    Win32ErrorCodes.ERROR_DS_GLOBAL_CANT_HAVE_LOCAL_MEMBER:
        Win32ErrorCodeDescription := 'A global group cannot have a local group as a member.';
    Win32ErrorCodes.ERROR_DS_GLOBAL_CANT_HAVE_UNIVERSAL_MEMBER:
        Win32ErrorCodeDescription := 'A global group cannot have a universal group as a member.';
    Win32ErrorCodes.ERROR_DS_UNIVERSAL_CANT_HAVE_LOCAL_MEMBER:
        Win32ErrorCodeDescription := 'A universal group cannot have a local group as a member.';
    Win32ErrorCodes.ERROR_DS_GLOBAL_CANT_HAVE_CROSSDOMAIN_MEMBER:
        Win32ErrorCodeDescription := 'A global group cannot have a cross-domain member.';
    Win32ErrorCodes.ERROR_DS_LOCAL_CANT_HAVE_CROSSDOMAIN_LOCAL_MEMBER:
        Win32ErrorCodeDescription :=
            'A local group cannot have another cross-domain local group as a member.';
    Win32ErrorCodes.ERROR_DS_HAVE_PRIMARY_MEMBERS:
        Win32ErrorCodeDescription :=
            'A group with primary members cannot change to a security-disabled group.';
    Win32ErrorCodes.ERROR_DS_STRING_SD_CONVERSION_FAILED:
        Win32ErrorCodeDescription :=
            'The schema cache load failed to convert the string default SD on a class-schema object.';
    Win32ErrorCodes.ERROR_DS_NAMING_MASTER_GC:
        Win32ErrorCodeDescription := 'Only DSAs configured to be Global Catalog servers should be allowed to hold the Domain Naming Master FSMO role. (Applies only to Windows 2000 servers)';
    Win32ErrorCodes.ERROR_DS_LOOKUP_FAILURE:
        Win32ErrorCodeDescription :=
            'The DSA operation is unable to proceed because of a DNS lookup failure.';
    Win32ErrorCodes.ERROR_DS_COULDNT_UPDATE_SPNS:
        Win32ErrorCodeDescription := 'While processing a change to the DNS Host Name for an object, the Service Principal Name values could not be kept in sync.';
    Win32ErrorCodes.ERROR_DS_CANT_RETRIEVE_SD:
        Win32ErrorCodeDescription := 'The Security Descriptor attribute could not be read.';
    Win32ErrorCodes.ERROR_DS_KEY_NOT_UNIQUE:
        Win32ErrorCodeDescription :=
            'The object requested was not found, but an object with that key was found.';
    Win32ErrorCodes.ERROR_DS_WRONG_LINKED_ATT_SYNTAX:
        Win32ErrorCodeDescription := 'The syntax of the linked attributed being added is incorrect. Forward links can only have syntax 2.5.5.1, 2.5.5.7, and 2.5.5.14, and backlinks can only have syntax 2.5.5.1.';
    Win32ErrorCodes.ERROR_DS_SAM_NEED_BOOTKEY_PASSWORD:
        Win32ErrorCodeDescription := 'Security Account Manager needs to get the boot password.';
    Win32ErrorCodes.ERROR_DS_SAM_NEED_BOOTKEY_FLOPPY:
        Win32ErrorCodeDescription :=
            'Security Account Manager needs to get the boot key from floppy disk.';
    Win32ErrorCodes.ERROR_DS_CANT_START:
        Win32ErrorCodeDescription := 'Directory Service cannot start.';
    Win32ErrorCodes.ERROR_DS_INIT_FAILURE:
        Win32ErrorCodeDescription := 'Directory Services could not start.';
    Win32ErrorCodes.ERROR_DS_NO_PKT_PRIVACY_ON_CONNECTION:
        Win32ErrorCodeDescription :=
            'The connection between client and server requires packet privacy or better.';
    Win32ErrorCodes.ERROR_DS_SOURCE_DOMAIN_IN_FOREST:
        Win32ErrorCodeDescription :=
            'The source domain may not be in the same forest as destination.';
    Win32ErrorCodes.ERROR_DS_DESTINATION_DOMAIN_NOT_IN_FOREST:
        Win32ErrorCodeDescription := 'The destination domain must be in the forest.';
    Win32ErrorCodes.ERROR_DS_DESTINATION_AUDITING_NOT_ENABLED:
        Win32ErrorCodeDescription :=
            'The operation requires that destination domain auditing be enabled.';
    Win32ErrorCodes.ERROR_DS_CANT_FIND_DC_FOR_SRC_DOMAIN:
        Win32ErrorCodeDescription := 'The operation couldnt locate a DC for the source domain.';
    Win32ErrorCodes.ERROR_DS_SRC_OBJ_NOT_GROUP_OR_USER:
        Win32ErrorCodeDescription := 'The source object must be a group or user.';
    Win32ErrorCodes.ERROR_DS_SRC_SID_EXISTS_IN_FOREST:
        Win32ErrorCodeDescription :=
            'The source objects SID already exists in destination forest.';
    Win32ErrorCodes.ERROR_DS_SRC_AND_DST_OBJECT_CLASS_MISMATCH:
        Win32ErrorCodeDescription := 'The source and destination object must be of the same type.';
    Win32ErrorCodes.ERROR_SAM_INIT_FAILURE:
        Win32ErrorCodeDescription := 'Security Accounts Manager initialization failed because of the following error: %1. Error Status: 0x%2. Click OK to shut down the system and reboot into Safe Mode. Check the event log for detailed information.';
    Win32ErrorCodes.ERROR_DS_DRA_SCHEMA_INFO_SHIP:
        Win32ErrorCodeDescription :=
            'Schema information could not be included in the replication request.';
    Win32ErrorCodes.ERROR_DS_DRA_SCHEMA_CONFLICT:
        Win32ErrorCodeDescription :=
            'The replication operation could not be completed due to a schema incompatibility.';
    Win32ErrorCodes.ERROR_DS_DRA_EARLIER_SCHEMA_CONLICT:
        Win32ErrorCodeDescription := 'The replication operation could not be completed due to a previous schema incompatibility.';
    Win32ErrorCodes.ERROR_DS_DRA_OBJ_NC_MISMATCH:
        Win32ErrorCodeDescription := 'The replication update could not be applied because either the source or the destination has not yet received information regarding a recent cross-domain move operation.';
    Win32ErrorCodes.ERROR_DS_NC_STILL_HAS_DSAS:
        Win32ErrorCodeDescription := 'The requested domain could not be deleted because there exist domain controllers that still host this domain.';
    Win32ErrorCodes.ERROR_DS_GC_REQUIRED:
        Win32ErrorCodeDescription :=
            'The requested operation can be performed only on a global catalog server.';
    Win32ErrorCodes.ERROR_DS_LOCAL_MEMBER_OF_LOCAL_ONLY:
        Win32ErrorCodeDescription :=
            'A local group can only be a member of other local groups in the same domain.';
    Win32ErrorCodes.ERROR_DS_NO_FPO_IN_UNIVERSAL_GROUPS:
        Win32ErrorCodeDescription :=
            'Foreign security principals cannot be members of universal groups.';
    Win32ErrorCodes.ERROR_DS_CANT_ADD_TO_GC:
        Win32ErrorCodeDescription :=
            'The attribute is not allowed to be replicated to the GC because of security reasons.';
    Win32ErrorCodes.ERROR_DS_NO_CHECKPOINT_WITH_PDC:
        Win32ErrorCodeDescription := 'The checkpoint with the PDC could not be taken because there are too many modifications being processed currently.';
    Win32ErrorCodes.ERROR_DS_SOURCE_AUDITING_NOT_ENABLED:
        Win32ErrorCodeDescription :=
            'The operation requires that source domain auditing be enabled.';
    Win32ErrorCodes.ERROR_DS_CANT_CREATE_IN_NONDOMAIN_NC:
        Win32ErrorCodeDescription :=
            'Security principal objects can only be created inside domain naming contexts.';
    Win32ErrorCodes.ERROR_DS_INVALID_NAME_FOR_SPN:
        Win32ErrorCodeDescription := 'A Service Principal Name (SPN) could not be constructed because the provided hostname is not in the necessary format.';
    Win32ErrorCodes.ERROR_DS_FILTER_USES_CONTRUCTED_ATTRS:
        Win32ErrorCodeDescription := 'A Filter was passed that uses constructed attributes.';
    Win32ErrorCodes.ERROR_DS_UNICODEPWD_NOT_IN_QUOTES:
        Win32ErrorCodeDescription :=
            'The unicodePwd attribute value must be enclosed in double quotes.';
    Win32ErrorCodes.ERROR_DS_MACHINE_ACCOUNT_QUOTA_EXCEEDED:
        Win32ErrorCodeDescription := 'Your computer could not be joined to the domain. You have exceeded the maximum number of computer accounts you are allowed to create in this domain. Contact your system administrator to have this limit reset or increased.';
    Win32ErrorCodes.ERROR_DS_MUST_BE_RUN_ON_DST_DC:
        Win32ErrorCodeDescription :=
            'For security reasons, the operation must be run on the destination DC.';
    Win32ErrorCodes.ERROR_DS_SRC_DC_MUST_BE_SP4_OR_GREATER:
        Win32ErrorCodeDescription :=
            'For security reasons, the source DC must be NT4SP4 or greater.';
    Win32ErrorCodes.ERROR_DS_CANT_TREE_DELETE_CRITICAL_OBJ:
        Win32ErrorCodeDescription := 'Critical Directory Service System objects cannot be deleted during tree delete operations. The tree delete may have been partially performed.';
    Win32ErrorCodes.ERROR_DS_INIT_FAILURE_CONSOLE:
        Win32ErrorCodeDescription := 'Directory Services could not start because of the following error: %1. Error Status: 0x%2. Please click OK to shutdown the system. You can use the recovery console to diagnose the system further.';
    Win32ErrorCodes.ERROR_DS_SAM_INIT_FAILURE_CONSOLE:
        Win32ErrorCodeDescription := 'Security Accounts Manager initialization failed because of the following error: %1. Error Status: 0x%2. Please click OK to shutdown the system. You can use the recovery console to diagnose the system further.';
    Win32ErrorCodes.ERROR_DS_FOREST_VERSION_TOO_HIGH:
        Win32ErrorCodeDescription := 'This version of Windows is too old to support the current directory forest behavior. You must upgrade the operating system on this server before it can become a domain controller in this forest.';
    Win32ErrorCodes.ERROR_DS_DOMAIN_VERSION_TOO_HIGH:
        Win32ErrorCodeDescription := 'This version of Windows is too old to support the current domain behavior. You must upgrade the operating system on this server before it can become a domain controller in this domain.';
    Win32ErrorCodes.ERROR_DS_FOREST_VERSION_TOO_LOW:
        Win32ErrorCodeDescription := 'This version of Windows no longer supports the behavior version in use in this directory forest. You must advance the forest behavior version before this server can become a domain controller in the forest.';
    Win32ErrorCodes.ERROR_DS_DOMAIN_VERSION_TOO_LOW:
        Win32ErrorCodeDescription := 'This version of Windows no longer supports the behavior version in use in this domain. You must advance the domain behavior version before this server can become a domain controller in the domain.';
    Win32ErrorCodes.ERROR_DS_INCOMPATIBLE_VERSION:
        Win32ErrorCodeDescription :=
            'The version of Windows is incompatible with the behavior version of the domain or forest.';
    Win32ErrorCodes.ERROR_DS_LOW_DSA_VERSION:
        Win32ErrorCodeDescription := 'The behavior version cannot be increased to the requested value because Domain Controllers still exist with versions lower than the requested value.';
    Win32ErrorCodes.ERROR_DS_NO_BEHAVIOR_VERSION_IN_MIXEDDOMAIN:
        Win32ErrorCodeDescription := 'The behavior version value cannot be increased while the domain is still in mixed domain mode. You must first change the domain to native mode before increasing the behavior version.';
    Win32ErrorCodes.ERROR_DS_NOT_SUPPORTED_SORT_ORDER:
        Win32ErrorCodeDescription := 'The sort order requested is not supported.';
    Win32ErrorCodes.ERROR_DS_NAME_NOT_UNIQUE:
        Win32ErrorCodeDescription := 'Found an object with a non unique name.';
    Win32ErrorCodes.ERROR_DS_MACHINE_ACCOUNT_CREATED_PRENT4:
        Win32ErrorCodeDescription :=
            'The machine account was created pre-NT4. The account needs to be recreated.';
    Win32ErrorCodes.ERROR_DS_OUT_OF_VERSION_STORE:
        Win32ErrorCodeDescription := 'The database is out of version store.';
    Win32ErrorCodes.ERROR_DS_INCOMPATIBLE_CONTROLS_USED:
        Win32ErrorCodeDescription :=
            'Unable to continue operation because multiple conflicting controls were used.';
    Win32ErrorCodes.ERROR_DS_NO_REF_DOMAIN:
        Win32ErrorCodeDescription :=
            'Unable to find a valid security descriptor reference domain for this partition.';
    Win32ErrorCodes.ERROR_DS_RESERVED_LINK_ID:
        Win32ErrorCodeDescription := 'Schema update failed: The link identifier is reserved.';
    Win32ErrorCodes.ERROR_DS_LINK_ID_NOT_AVAILABLE:
        Win32ErrorCodeDescription :=
            'Schema update failed: There are no link identifiers available.';
    Win32ErrorCodes.ERROR_DS_AG_CANT_HAVE_UNIVERSAL_MEMBER:
        Win32ErrorCodeDescription :=
            'An account group can not have a universal group as a member.';
    Win32ErrorCodes.ERROR_DS_MODIFYDN_DISALLOWED_BY_INSTANCE_TYPE:
        Win32ErrorCodeDescription :=
            'Rename or move operations on naming context heads or read-only objects are not allowed.';
    Win32ErrorCodes.ERROR_DS_NO_OBJECT_MOVE_IN_SCHEMA_NC:
        Win32ErrorCodeDescription :=
            'Move operations on objects in the schema naming context are not allowed.';
    Win32ErrorCodes.ERROR_DS_MODIFYDN_DISALLOWED_BY_FLAG:
        Win32ErrorCodeDescription := 'A system flag has been set on the object and does not allow the object to be moved or renamed.';
    Win32ErrorCodes.ERROR_DS_MODIFYDN_WRONG_GRANDPARENT:
        Win32ErrorCodeDescription := 'This object is not allowed to change its grandparent container. Moves are not forbidden on this object, but are restricted to sibling containers.';
    Win32ErrorCodes.ERROR_DS_NAME_ERROR_TRUST_REFERRAL:
        Win32ErrorCodeDescription :=
            'Unable to resolve completely, a referral to another forest is generated.';
    Win32ErrorCodes.ERROR_NOT_SUPPORTED_ON_STANDARD_SERVER:
        Win32ErrorCodeDescription := 'The requested action is not supported on standard server.';
    Win32ErrorCodes.ERROR_DS_CANT_ACCESS_REMOTE_PART_OF_AD:
        Win32ErrorCodeDescription := 'Could not access a partition of the Active Directory located on a remote server. Make sure at least one server is running for the partition in question.';
    Win32ErrorCodes.ERROR_DS_CR_IMPOSSIBLE_TO_VALIDATE_V2:
        Win32ErrorCodeDescription := 'The directory cant validate the proposed naming context (or partition) name because it doesnt hold a replica nor can it contact a replica of the naming context above the proposed naming context.';
    Win32ErrorCodes.ERROR_DS_THREAD_LIMIT_EXCEEDED:
        Win32ErrorCodeDescription := 'The thread limit for this request was exceeded.';
    Win32ErrorCodes.ERROR_DS_NOT_CLOSEST:
        Win32ErrorCodeDescription := 'The Global catalog server is not in the closet site.';
    Win32ErrorCodes.DNS_ERROR_RCODE_FORMAT_ERROR:
        Win32ErrorCodeDescription := 'DNS server unable to interpret format.';
    Win32ErrorCodes.DNS_ERROR_RCODE_SERVER_FAILURE:
        Win32ErrorCodeDescription := 'DNS server failure.';
    Win32ErrorCodes.DNS_ERROR_RCODE_NAME_ERROR:
        Win32ErrorCodeDescription := 'DNS name does not exist.';
    Win32ErrorCodes.DNS_ERROR_RCODE_NOT_IMPLEMENTED:
        Win32ErrorCodeDescription := 'DNS request not supported by name server.';
    Win32ErrorCodes.DNS_ERROR_RCODE_REFUSED:
        Win32ErrorCodeDescription := 'DNS operation refused.';
    Win32ErrorCodes.DNS_ERROR_RCODE_YXDOMAIN:
        Win32ErrorCodeDescription := 'DNS name that ought not exist, does exist.';
    Win32ErrorCodes.DNS_ERROR_RCODE_YXRRSET:
        Win32ErrorCodeDescription := 'DNS RR set that ought not exist, does exist.';
    Win32ErrorCodes.DNS_ERROR_RCODE_NXRRSET:
        Win32ErrorCodeDescription := 'DNS RR set that ought to exist, does not exist.';
    Win32ErrorCodes.DNS_ERROR_RCODE_NOTAUTH:
        Win32ErrorCodeDescription := 'DNS server not authoritative for zone.';
    Win32ErrorCodes.DNS_ERROR_RCODE_NOTZONE:
        Win32ErrorCodeDescription := 'DNS name in update or prereq is not in zone.';
    Win32ErrorCodes.DNS_ERROR_RCODE_BADSIG:
        Win32ErrorCodeDescription := 'DNS signature failed to verify.';
    Win32ErrorCodes.DNS_ERROR_RCODE_BADKEY:
        Win32ErrorCodeDescription := 'DNS bad key.';
    Win32ErrorCodes.DNS_ERROR_RCODE_BADTIME:
        Win32ErrorCodeDescription := 'DNS signature validity expired.';
    Win32ErrorCodes.DNS_INFO_NO_RECORDS:
        Win32ErrorCodeDescription := 'No records found for given DNS query.';
    Win32ErrorCodes.DNS_ERROR_BAD_PACKET:
        Win32ErrorCodeDescription := 'Bad DNS packet.';
    Win32ErrorCodes.DNS_ERROR_NO_PACKET:
        Win32ErrorCodeDescription := 'No DNS packet.';
    Win32ErrorCodes.DNS_ERROR_RCODE:
        Win32ErrorCodeDescription := 'DNS error, check rcode.';
    Win32ErrorCodes.DNS_ERROR_UNSECURE_PACKET:
        Win32ErrorCodeDescription := 'Unsecured DNS packet.';
    Win32ErrorCodes.DNS_ERROR_INVALID_TYPE:
        Win32ErrorCodeDescription := 'Invalid DNS type.';
    Win32ErrorCodes.DNS_ERROR_INVALID_IP_ADDRESS:
        Win32ErrorCodeDescription := 'Invalid IP address.';
    Win32ErrorCodes.DNS_ERROR_INVALID_PROPERTY:
        Win32ErrorCodeDescription := 'Invalid property.';
    Win32ErrorCodes.DNS_ERROR_TRY_AGAIN_LATER:
        Win32ErrorCodeDescription := 'Try DNS operation again later.';
    Win32ErrorCodes.DNS_ERROR_NOT_UNIQUE:
        Win32ErrorCodeDescription := 'Record for given name and type is not unique.';
    Win32ErrorCodes.DNS_ERROR_NON_RFC_NAME:
        Win32ErrorCodeDescription := 'DNS name does not comply with RFC specifications.';
    Win32ErrorCodes.DNS_STATUS_FQDN:
        Win32ErrorCodeDescription := 'DNS name is a fully-qualified DNS name.';
    Win32ErrorCodes.DNS_STATUS_DOTTED_NAME:
        Win32ErrorCodeDescription := 'DNS name is dotted (multi-label).';
    Win32ErrorCodes.DNS_STATUS_SINGLE_PART_NAME:
        Win32ErrorCodeDescription := 'DNS name is a single-part name.';
    Win32ErrorCodes.DNS_ERROR_INVALID_NAME_CHAR:
        Win32ErrorCodeDescription := 'DSN name contains an invalid character.';
    Win32ErrorCodes.DNS_ERROR_NUMERIC_NAME:
        Win32ErrorCodeDescription := 'DNS name is entirely numeric.';
    Win32ErrorCodes.DNS_ERROR_ZONE_DOES_NOT_EXIST:
        Win32ErrorCodeDescription := 'DNS zone does not exist.';
    Win32ErrorCodes.DNS_ERROR_NO_ZONE_INFO:
        Win32ErrorCodeDescription := 'DNS zone information not available.';
    Win32ErrorCodes.DNS_ERROR_INVALID_ZONE_OPERATION:
        Win32ErrorCodeDescription := 'Invalid operation for DNS zone.';
    Win32ErrorCodes.DNS_ERROR_ZONE_CONFIGURATION_ERROR:
        Win32ErrorCodeDescription := 'Invalid DNS zone configuration.';
    Win32ErrorCodes.DNS_ERROR_ZONE_HAS_NO_SOA_RECORD:
        Win32ErrorCodeDescription := 'DNS zone has no start of authority (SOA) record.';
    Win32ErrorCodes.DNS_ERROR_ZONE_HAS_NO_NS_RECORDS:
        Win32ErrorCodeDescription := 'DNS zone has no name server (NS) record.';
    Win32ErrorCodes.DNS_ERROR_ZONE_LOCKED:
        Win32ErrorCodeDescription := 'DNS zone is locked.';
    Win32ErrorCodes.DNS_ERROR_ZONE_CREATION_FAILED:
        Win32ErrorCodeDescription := 'DNS zone creation failed.';
    Win32ErrorCodes.DNS_ERROR_ZONE_ALREADY_EXISTS:
        Win32ErrorCodeDescription := 'DNS zone already exists.';
    Win32ErrorCodes.DNS_ERROR_AUTOZONE_ALREADY_EXISTS:
        Win32ErrorCodeDescription := 'DNS automatic zone already exists.';
    Win32ErrorCodes.DNS_ERROR_INVALID_ZONE_TYPE:
        Win32ErrorCodeDescription := 'Invalid DNS zone type.';
    Win32ErrorCodes.DNS_ERROR_SECONDARY_REQUIRES_MASTER_IP:
        Win32ErrorCodeDescription := 'Secondary DNS zone requires master IP address.';
    Win32ErrorCodes.DNS_ERROR_ZONE_NOT_SECONDARY:
        Win32ErrorCodeDescription := 'DNS zone not secondary.';
    Win32ErrorCodes.DNS_ERROR_NEED_SECONDARY_ADDRESSES:
        Win32ErrorCodeDescription := 'Need secondary IP address.';
    Win32ErrorCodes.DNS_ERROR_WINS_INIT_FAILED:
        Win32ErrorCodeDescription := 'WINS initialization failed.';
    Win32ErrorCodes.DNS_ERROR_NEED_WINS_SERVERS:
        Win32ErrorCodeDescription := 'Need WINS servers.';
    Win32ErrorCodes.DNS_ERROR_NBSTAT_INIT_FAILED:
        Win32ErrorCodeDescription := 'NBTSTAT initialization call failed.';
    Win32ErrorCodes.DNS_ERROR_SOA_DELETE_INVALID:
        Win32ErrorCodeDescription := 'Invalid delete of start of authority (SOA)';
    Win32ErrorCodes.DNS_ERROR_FORWARDER_ALREADY_EXISTS:
        Win32ErrorCodeDescription := 'A conditional forwarding zone already exists for that name.';
    Win32ErrorCodes.DNS_ERROR_PRIMARY_REQUIRES_DATAFILE:
        Win32ErrorCodeDescription := 'Primary DNS zone requires datafile.';
    Win32ErrorCodes.DNS_ERROR_INVALID_DATAFILE_NAME:
        Win32ErrorCodeDescription := 'Invalid datafile name for DNS zone.';
    Win32ErrorCodes.DNS_ERROR_DATAFILE_OPEN_FAILURE:
        Win32ErrorCodeDescription := 'Failed to open datafile for DNS zone.';
    Win32ErrorCodes.DNS_ERROR_FILE_WRITEBACK_FAILED:
        Win32ErrorCodeDescription := 'Failed to write datafile for DNS zone.';
    Win32ErrorCodes.DNS_ERROR_DATAFILE_PARSING:
        Win32ErrorCodeDescription := 'Failure while reading datafile for DNS zone.';
    Win32ErrorCodes.DNS_ERROR_RECORD_DOES_NOT_EXIST:
        Win32ErrorCodeDescription := 'DNS record does not exist.';
    Win32ErrorCodes.DNS_ERROR_RECORD_FORMAT:
        Win32ErrorCodeDescription := 'DNS record format error.';
    Win32ErrorCodes.DNS_ERROR_NODE_CREATION_FAILED:
        Win32ErrorCodeDescription := 'Node creation failure in DNS.';
    Win32ErrorCodes.DNS_ERROR_UNKNOWN_RECORD_TYPE:
        Win32ErrorCodeDescription := 'Unknown DNS record type.';
    Win32ErrorCodes.DNS_ERROR_RECORD_TIMED_OUT:
        Win32ErrorCodeDescription := 'DNS record timed out.';
    Win32ErrorCodes.DNS_ERROR_NAME_NOT_IN_ZONE:
        Win32ErrorCodeDescription := 'Name not in DNS zone.';
    Win32ErrorCodes.DNS_ERROR_CNAME_LOOP:
        Win32ErrorCodeDescription := 'CNAME loop detected.';
    Win32ErrorCodes.DNS_ERROR_NODE_IS_CNAME:
        Win32ErrorCodeDescription := 'Node is a CNAME DNS record.';
    Win32ErrorCodes.DNS_ERROR_CNAME_COLLISION:
        Win32ErrorCodeDescription := 'A CNAME record already exists for given name.';
    Win32ErrorCodes.DNS_ERROR_RECORD_ONLY_AT_ZONE_ROOT:
        Win32ErrorCodeDescription := 'Record only at DNS zone root.';
    Win32ErrorCodes.DNS_ERROR_RECORD_ALREADY_EXISTS:
        Win32ErrorCodeDescription := 'DNS record already exists.';
    Win32ErrorCodes.DNS_ERROR_SECONDARY_DATA:
        Win32ErrorCodeDescription := 'Secondary DNS zone data error.';
    Win32ErrorCodes.DNS_ERROR_NO_CREATE_CACHE_DATA:
        Win32ErrorCodeDescription := 'Could not create DNS cache data.';
    Win32ErrorCodes.DNS_ERROR_NAME_DOES_NOT_EXIST:
        Win32ErrorCodeDescription := 'DNS name does not exist.';
    Win32ErrorCodes.DNS_WARNING_PTR_CREATE_FAILED:
        Win32ErrorCodeDescription := 'Could not create pointer (PTR) record.';
    Win32ErrorCodes.DNS_WARNING_DOMAIN_UNDELETED:
        Win32ErrorCodeDescription := 'DNS domain was undeleted.';
    Win32ErrorCodes.DNS_ERROR_DS_UNAVAILABLE:
        Win32ErrorCodeDescription := 'The directory service is unavailable.';
    Win32ErrorCodes.DNS_ERROR_DS_ZONE_ALREADY_EXISTS:
        Win32ErrorCodeDescription := 'DNS zone already exists in the directory service.';
    Win32ErrorCodes.DNS_ERROR_NO_BOOTFILE_IF_DS_ZONE:
        Win32ErrorCodeDescription := 'DNS server not creating or reading the boot file for the directory service integrated DNS zone.';
    Win32ErrorCodes.DNS_INFO_AXFR_COMPLETE:
        Win32ErrorCodeDescription := 'DNS AXFR (zone transfer) complete.';
    Win32ErrorCodes.DNS_ERROR_AXFR:
        Win32ErrorCodeDescription := 'DNS zone transfer failed.';
    Win32ErrorCodes.DNS_INFO_ADDED_LOCAL_WINS:
        Win32ErrorCodeDescription := 'Added local WINS server.';
    Win32ErrorCodes.DNS_STATUS_CONTINUE_NEEDED:
        Win32ErrorCodeDescription := 'Secure update call needs to continue update request.';
    Win32ErrorCodes.DNS_ERROR_NO_TCPIP:
        Win32ErrorCodeDescription := 'TCP/IP network protocol not installed.';
    Win32ErrorCodes.DNS_ERROR_NO_DNS_SERVERS:
        Win32ErrorCodeDescription := 'No DNS servers configured for local system.';
    Win32ErrorCodes.DNS_ERROR_DP_DOES_NOT_EXIST:
        Win32ErrorCodeDescription := 'The specified directory partition does not exist.';
    Win32ErrorCodes.DNS_ERROR_DP_ALREADY_EXISTS:
        Win32ErrorCodeDescription := 'The specified directory partition already exists.';
    Win32ErrorCodes.DNS_ERROR_DP_NOT_ENLISTED:
        Win32ErrorCodeDescription :=
            'The DS is not enlisted in the specified directory partition.';
    Win32ErrorCodes.DNS_ERROR_DP_ALREADY_ENLISTED:
        Win32ErrorCodeDescription :=
            'The DS is already enlisted in the specified directory partition.';
    Win32ErrorCodes.WSAEINTR:
        Win32ErrorCodeDescription :=
            'A blocking operation was interrupted by a call to WSACancelBlockingCall.';
    Win32ErrorCodes.WSAEBADF:
        Win32ErrorCodeDescription := 'The file handle supplied is not valid.';
    Win32ErrorCodes.WSAEACCES:
        Win32ErrorCodeDescription :=
            'An attempt was made to access a socket in a way forbidden by its access permissions.';
    Win32ErrorCodes.WSAEFAULT:
        Win32ErrorCodeDescription := 'The system detected an invalid pointer address in attempting to use a pointer argument in a call.';
    Win32ErrorCodes.WSAEINVAL:
        Win32ErrorCodeDescription := 'An invalid argument was supplied.';
    Win32ErrorCodes.WSAEMFILE:
        Win32ErrorCodeDescription := 'Too many open sockets.';
    Win32ErrorCodes.WSAEWOULDBLOCK:
        Win32ErrorCodeDescription :=
            'A non-blocking socket operation could not be completed immediately.';
    Win32ErrorCodes.WSAEINPROGRESS:
        Win32ErrorCodeDescription := 'A blocking operation is currently executing.';
    Win32ErrorCodes.WSAEALREADY:
        Win32ErrorCodeDescription := 'An operation was attempted on a non-blocking socket that already had an operation in progress.';
    Win32ErrorCodes.WSAENOTSOCK:
        Win32ErrorCodeDescription :=
            'An operation was attempted on something that is not a socket.';
    Win32ErrorCodes.WSAEDESTADDRREQ:
        Win32ErrorCodeDescription :=
            'A required address was omitted from an operation on a socket.';
    Win32ErrorCodes.WSAEMSGSIZE:
        Win32ErrorCodeDescription := 'A message sent on a datagram socket was larger than the internal message buffer or some other network limit, or the buffer used to receive a datagram into was smaller than the datagram itself.';
    Win32ErrorCodes.WSAEPROTOTYPE:
        Win32ErrorCodeDescription := 'A protocol was specified in the socket function call that does not support the semantics of the socket type requested.';
    Win32ErrorCodes.WSAENOPROTOOPT:
        Win32ErrorCodeDescription := 'An unknown, invalid, or unsupported option or level was specified in a getsockopt or setsockopt call.';
    Win32ErrorCodes.WSAEPROTONOSUPPORT:
        Win32ErrorCodeDescription := 'The requested protocol has not been configured into the system, or no implementation for it exists.';
    Win32ErrorCodes.WSAESOCKTNOSUPPORT:
        Win32ErrorCodeDescription :=
            'The support for the specified socket type does not exist in this address family.';
    Win32ErrorCodes.WSAEOPNOTSUPP:
        Win32ErrorCodeDescription :=
            'The attempted operation is not supported for the type of object referenced.';
    Win32ErrorCodes.WSAEPFNOSUPPORT:
        Win32ErrorCodeDescription := 'The protocol family has not been configured into the system or no implementation for it exists.';
    Win32ErrorCodes.WSAEAFNOSUPPORT:
        Win32ErrorCodeDescription :=
            'An address incompatible with the requested protocol was used.';
    Win32ErrorCodes.WSAEADDRINUSE:
        Win32ErrorCodeDescription := 'Only one usage of each socket address (protocol/network address/port) is normally permitted.';
    Win32ErrorCodes.WSAEADDRNOTAVAIL:
        Win32ErrorCodeDescription := 'The requested address is not valid in its context.';
    Win32ErrorCodes.WSAENETDOWN:
        Win32ErrorCodeDescription := 'A socket operation encountered a dead network.';
    Win32ErrorCodes.WSAENETUNREACH:
        Win32ErrorCodeDescription := 'A socket operation was attempted to an unreachable network.';
    Win32ErrorCodes.WSAENETRESET:
        Win32ErrorCodeDescription := 'The connection has been broken due to keep-alive activity detecting a failure while the operation was in progress.';
    Win32ErrorCodes.WSAECONNABORTED:
        Win32ErrorCodeDescription :=
            'An established connection was aborted by the software in your host machine.';
    Win32ErrorCodes.WSAECONNRESET:
        Win32ErrorCodeDescription :=
            'An existing connection was forcibly closed by the remote host.';
    Win32ErrorCodes.WSAENOBUFS:
        Win32ErrorCodeDescription := 'An operation on a socket could not be performed because the system lacked sufficient buffer space or because a queue was full.';
    Win32ErrorCodes.WSAEISCONN:
        Win32ErrorCodeDescription := 'A connect request was made on an already connected socket.';
    Win32ErrorCodes.WSAENOTCONN:
        Win32ErrorCodeDescription := 'A request to send or receive data was disallowed because the socket is not connected and (when sending on a datagram socket using a sendto call) no address was supplied.';
    Win32ErrorCodes.WSAESHUTDOWN:
        Win32ErrorCodeDescription := 'A request to send or receive data was disallowed because the socket had already been shut down in that direction with a previous shutdown call.';
    Win32ErrorCodes.WSAETOOMANYREFS:
        Win32ErrorCodeDescription := 'Too many references to some kernel object.';
    Win32ErrorCodes.WSAETIMEDOUT:
        Win32ErrorCodeDescription := 'A connection attempt failed because the connected party did not properly respond after a period of time, or established connection failed because connected host has failed to respond.';
    Win32ErrorCodes.WSAECONNREFUSED:
        Win32ErrorCodeDescription :=
            'No connection could be made because the target machine actively refused it.';
    Win32ErrorCodes.WSAELOOP:
        Win32ErrorCodeDescription := 'Cannot translate name.';
    Win32ErrorCodes.WSAENAMETOOLONG:
        Win32ErrorCodeDescription := 'Name component or name was too long.';
    Win32ErrorCodes.WSAEHOSTDOWN:
        Win32ErrorCodeDescription :=
            'A socket operation failed because the destination host was down.';
    Win32ErrorCodes.WSAEHOSTUNREACH:
        Win32ErrorCodeDescription := 'A socket operation was attempted to an unreachable host.';
    Win32ErrorCodes.WSAENOTEMPTY:
        Win32ErrorCodeDescription := 'Cannot remove a directory that is not empty.';
    Win32ErrorCodes.WSAEPROCLIM:
        Win32ErrorCodeDescription := 'A Windows Sockets implementation may have a limit on the number of applications that may use it simultaneously.';
    Win32ErrorCodes.WSAEUSERS:
        Win32ErrorCodeDescription := 'Ran out of quota.';
    Win32ErrorCodes.WSAEDQUOT:
        Win32ErrorCodeDescription := 'Ran out of disk quota.';
    Win32ErrorCodes.WSAESTALE:
        Win32ErrorCodeDescription := 'File handle reference is no longer available.';
    Win32ErrorCodes.WSAEREMOTE:
        Win32ErrorCodeDescription := 'Item is not available locally.';
    Win32ErrorCodes.WSASYSNOTREADY:
        Win32ErrorCodeDescription := 'WSAStartup cannot function at this time because the underlying system it uses to provide network services is currently unavailable.';
    Win32ErrorCodes.WSAVERNOTSUPPORTED:
        Win32ErrorCodeDescription := 'The Windows Sockets version requested is not supported.';
    Win32ErrorCodes.WSANOTINITIALISED:
        Win32ErrorCodeDescription :=
            'Either the application has not called WSAStartup, or WSAStartup failed.';
    Win32ErrorCodes.WSAEDISCON:
        Win32ErrorCodeDescription := 'Returned by WSARecv or WSARecvFrom to indicate the remote party has initiated a graceful shutdown sequence.';
    Win32ErrorCodes.WSAENOMORE:
        Win32ErrorCodeDescription := 'No more results can be returned by WSALookupServiceNext.';
    Win32ErrorCodes.WSAECANCELLED:
        Win32ErrorCodeDescription := 'A call to WSALookupServiceEnd was made while this call was still processing. The call has been canceled.';
    Win32ErrorCodes.WSAEINVALIDPROCTABLE:
        Win32ErrorCodeDescription := 'The procedure call table is invalid.';
    Win32ErrorCodes.WSAEINVALIDPROVIDER:
        Win32ErrorCodeDescription := 'The requested service provider is invalid.';
    Win32ErrorCodes.WSAEPROVIDERFAILEDINIT:
        Win32ErrorCodeDescription :=
            'The requested service provider could not be loaded or initialized.';
    Win32ErrorCodes.WSASYSCALLFAILURE:
        Win32ErrorCodeDescription := 'A system call that should never fail has failed.';
    Win32ErrorCodes.WSASERVICE_NOT_FOUND:
        Win32ErrorCodeDescription :=
            'No such service is known. The service cannot be found in the specified name space.';
    Win32ErrorCodes.WSATYPE_NOT_FOUND:
        Win32ErrorCodeDescription := 'The specified class was not found.';
    Win32ErrorCodes.WSA_E_NO_MORE:
        Win32ErrorCodeDescription := 'No more results can be returned by WSALookupServiceNext.';
    Win32ErrorCodes.WSA_E_CANCELLED:
        Win32ErrorCodeDescription := 'A call to WSALookupServiceEnd was made while this call was still processing. The call has been canceled.';
    Win32ErrorCodes.WSAEREFUSED:
        Win32ErrorCodeDescription := 'A database query failed because it was actively refused.';
    Win32ErrorCodes.WSAHOST_NOT_FOUND:
        Win32ErrorCodeDescription := 'No such host is known.';
    Win32ErrorCodes.WSATRY_AGAIN:
        Win32ErrorCodeDescription := 'This is usually a temporary error during hostname resolution and means that the local server did not receive a response from an authoritative server.';
    Win32ErrorCodes.WSANO_RECOVERY:
        Win32ErrorCodeDescription := 'A non-recoverable error occurred during a database lookup.';
    Win32ErrorCodes.WSANO_DATA:
        Win32ErrorCodeDescription := 'The requested name is valid and was found in the database, but it does not have the correct associated data being resolved for.';
    Win32ErrorCodes.WSA_QOS_RECEIVERS:
        Win32ErrorCodeDescription := 'At least one reserve has arrived.';
    Win32ErrorCodes.WSA_QOS_SENDERS:
        Win32ErrorCodeDescription := 'At least one path has arrived.';
    Win32ErrorCodes.WSA_QOS_NO_SENDERS:
        Win32ErrorCodeDescription := 'There are no senders.';
    Win32ErrorCodes.WSA_QOS_NO_RECEIVERS:
        Win32ErrorCodeDescription := 'There are no receivers.';
    Win32ErrorCodes.WSA_QOS_REQUEST_CONFIRMED:
        Win32ErrorCodeDescription := 'Reserve has been confirmed.';
    Win32ErrorCodes.WSA_QOS_ADMISSION_FAILURE:
        Win32ErrorCodeDescription := 'Error due to lack of resources.';
    Win32ErrorCodes.WSA_QOS_POLICY_FAILURE:
        Win32ErrorCodeDescription := 'Rejected for administrative reasons - bad credentials.';
    Win32ErrorCodes.WSA_QOS_BAD_STYLE:
        Win32ErrorCodeDescription := 'Unknown or conflicting style.';
    Win32ErrorCodes.WSA_QOS_BAD_OBJECT:
        Win32ErrorCodeDescription :=
            'Problem with some part of the filterspec or providerspecific buffer in general.';
    Win32ErrorCodes.WSA_QOS_TRAFFIC_CTRL_ERROR:
        Win32ErrorCodeDescription := 'Problem with some part of the flowspec.';
    Win32ErrorCodes.WSA_QOS_GENERIC_ERROR:
        Win32ErrorCodeDescription := 'General QOS error.';
    Win32ErrorCodes.WSA_QOS_ESERVICETYPE:
        Win32ErrorCodeDescription :=
            'An invalid or unrecognized service type was found in the flowspec.';
    Win32ErrorCodes.WSA_QOS_EFLOWSPEC:
        Win32ErrorCodeDescription :=
            'An invalid or inconsistent flowspec was found in the QOS structure.';
    Win32ErrorCodes.WSA_QOS_EPROVSPECBUF:
        Win32ErrorCodeDescription := 'Invalid QOS provider-specific buffer.';
    Win32ErrorCodes.WSA_QOS_EFILTERSTYLE:
        Win32ErrorCodeDescription := 'An invalid QOS filter style was used.';
    Win32ErrorCodes.WSA_QOS_EFILTERTYPE:
        Win32ErrorCodeDescription := 'An invalid QOS filter type was used.';
    Win32ErrorCodes.WSA_QOS_EFILTERCOUNT:
        Win32ErrorCodeDescription :=
            'An incorrect number of QOS FILTERSPECs were specified in the FLOWDESCRIPTOR.';
    Win32ErrorCodes.WSA_QOS_EOBJLENGTH:
        Win32ErrorCodeDescription := 'An object with an invalid ObjectLength field was specified in the QOS provider-specific buffer.';
    Win32ErrorCodes.WSA_QOS_EFLOWCOUNT:
        Win32ErrorCodeDescription :=
            'An incorrect number of flow descriptors was specified in the QOS structure.';
    Win32ErrorCodes.WSA_QOS_EUNKNOWNPSOBJ:
        Win32ErrorCodeDescription :=
            'An unrecognized object was found in the QOS provider-specific buffer.';
    Win32ErrorCodes.WSA_QOS_EPOLICYOBJ:
        Win32ErrorCodeDescription :=
            'An invalid policy object was found in the QOS provider-specific buffer.';
    Win32ErrorCodes.WSA_QOS_EFLOWDESC:
        Win32ErrorCodeDescription :=
            'An invalid QOS flow descriptor was found in the flow descriptor list.';
    Win32ErrorCodes.WSA_QOS_EPSFLOWSPEC:
        Win32ErrorCodeDescription :=
            'An invalid or inconsistent flowspec was found in the QOS provider-specific buffer.';
    Win32ErrorCodes.WSA_QOS_EPSFILTERSPEC:
        Win32ErrorCodeDescription :=
            'An invalid FILTERSPEC was found in the QOS provider-specific buffer.';
    Win32ErrorCodes.WSA_QOS_ESDMODEOBJ:
        Win32ErrorCodeDescription :=
            'An invalid shape discard mode object was found in the QOS provider-specific buffer.';
    Win32ErrorCodes.WSA_QOS_ESHAPERATEOBJ:
        Win32ErrorCodeDescription :=
            'An invalid shaping rate object was found in the QOS provider-specific buffer.';
    Win32ErrorCodes.WSA_QOS_RESERVED_PETYPE:
        Win32ErrorCodeDescription :=
            'A reserved policy element was found in the QOS provider-specific buffer.';
    Win32ErrorCodes.ERROR_SXS_SECTION_NOT_FOUND:
        Win32ErrorCodeDescription :=
            'The requested section was not present in the activation context.';
    Win32ErrorCodes.ERROR_SXS_CANT_GEN_ACTCTX:
        Win32ErrorCodeDescription := 'This application has failed to start because the application configuration is incorrect. Reinstalling the application may fix this problem.';
    Win32ErrorCodes.ERROR_SXS_INVALID_ACTCTXDATA_FORMAT:
        Win32ErrorCodeDescription := 'The application binding data format is invalid.';
    Win32ErrorCodes.ERROR_SXS_ASSEMBLY_NOT_FOUND:
        Win32ErrorCodeDescription := 'The referenced assembly is not installed on your system.';
    Win32ErrorCodes.ERROR_SXS_MANIFEST_FORMAT_ERROR:
        Win32ErrorCodeDescription :=
            'The manifest file does not begin with the required tag and format information.';
    Win32ErrorCodes.ERROR_SXS_MANIFEST_PARSE_ERROR:
        Win32ErrorCodeDescription := 'The manifest file contains one or more syntax errors.';
    Win32ErrorCodes.ERROR_SXS_ACTIVATION_CONTEXT_DISABLED:
        Win32ErrorCodeDescription :=
            'The application attempted to activate a disabled activation context.';
    Win32ErrorCodes.ERROR_SXS_KEY_NOT_FOUND:
        Win32ErrorCodeDescription :=
            'The requested lookup key was not found in any active activation context.';
    Win32ErrorCodes.ERROR_SXS_VERSION_CONFLICT:
        Win32ErrorCodeDescription := 'A component version required by the application conflicts with another component version already active.';
    Win32ErrorCodes.ERROR_SXS_WRONG_SECTION_TYPE:
        Win32ErrorCodeDescription :=
            'The type requested activation context section does not match the query API used.';
    Win32ErrorCodes.ERROR_SXS_THREAD_QUERIES_DISABLED:
        Win32ErrorCodeDescription := 'Lack of system resources has required isolated activation to be disabled for the current thread of execution.';
    Win32ErrorCodes.ERROR_SXS_PROCESS_DEFAULT_ALREADY_SET:
        Win32ErrorCodeDescription := 'An attempt to set the process default activation context failed because the process default activation context was already set.';
    Win32ErrorCodes.ERROR_SXS_UNKNOWN_ENCODING_GROUP:
        Win32ErrorCodeDescription := 'The encoding group identifier specified is not recognized.';
    Win32ErrorCodes.ERROR_SXS_UNKNOWN_ENCODING:
        Win32ErrorCodeDescription := 'The encoding requested is not recognized.';
    Win32ErrorCodes.ERROR_SXS_INVALID_XML_NAMESPACE_URI:
        Win32ErrorCodeDescription := 'The manifest contains a reference to an invalid URI.';
    Win32ErrorCodes.ERROR_SXS_ROOT_MANIFEST_DEPENDENCY_NOT_INSTALLED:
        Win32ErrorCodeDescription := 'The application manifest contains a reference to a dependent assembly which is not installed.';
    Win32ErrorCodes.ERROR_SXS_LEAF_MANIFEST_DEPENDENCY_NOT_INSTALLED:
        Win32ErrorCodeDescription := 'The manifest for an assembly used by the application has a reference to a dependent assembly which is not installed.';
    Win32ErrorCodes.ERROR_SXS_INVALID_ASSEMBLY_IDENTITY_ATTRIBUTE:
        Win32ErrorCodeDescription :=
            'The manifest contains an attribute for the assembly identity which is not valid.';
    Win32ErrorCodes.ERROR_SXS_MANIFEST_MISSING_REQUIRED_DEFAULT_NAMESPACE:
        Win32ErrorCodeDescription := 'The manifest is missing the required default namespace specification on the assembly element.';
    Win32ErrorCodes.ERROR_SXS_MANIFEST_INVALID_REQUIRED_DEFAULT_NAMESPACE:
        Win32ErrorCodeDescription := 'The manifest has a default namespace specified on the assembly element but its value is not "urn:schemas-microsoft-com:asm.v1".';
    Win32ErrorCodes.ERROR_SXS_PRIVATE_MANIFEST_CROSS_PATH_WITH_REPARSE_POINT:
        Win32ErrorCodeDescription :=
            'The private manifest probe has crossed the reparse-point-associated path.';
    Win32ErrorCodes.ERROR_SXS_DUPLICATE_DLL_NAME:
        Win32ErrorCodeDescription := 'Two or more components referenced directly or indirectly by the application manifest have files by the same name.';
    Win32ErrorCodes.ERROR_SXS_DUPLICATE_WINDOWCLASS_NAME:
        Win32ErrorCodeDescription := 'Two or more components referenced directly or indirectly by the application manifest have window classes with the same name.';
    Win32ErrorCodes.ERROR_SXS_DUPLICATE_CLSID:
        Win32ErrorCodeDescription := 'Two or more components referenced directly or indirectly by the application manifest have the same COM server CLSIDs.';
    Win32ErrorCodes.ERROR_SXS_DUPLICATE_IID:
        Win32ErrorCodeDescription := 'Two or more components referenced directly or indirectly by the application manifest have proxies for the same COM interface IIDs.';
    Win32ErrorCodes.ERROR_SXS_DUPLICATE_TLBID:
        Win32ErrorCodeDescription := 'Two or more components referenced directly or indirectly by the application manifest have the same COM type library TLBIDs.';
    Win32ErrorCodes.ERROR_SXS_DUPLICATE_PROGID:
        Win32ErrorCodeDescription := 'Two or more components referenced directly or indirectly by the application manifest have the same COM ProgIDs.';
    Win32ErrorCodes.ERROR_SXS_DUPLICATE_ASSEMBLY_NAME:
        Win32ErrorCodeDescription := 'Two or more components referenced directly or indirectly by the application manifest are different versions of the same component which is not permitted.';
    Win32ErrorCodes.ERROR_SXS_FILE_HASH_MISMATCH:
        Win32ErrorCodeDescription := 'A components file does not match the verification information present in the component manifest.';
    Win32ErrorCodes.ERROR_SXS_POLICY_PARSE_ERROR:
        Win32ErrorCodeDescription := 'The policy manifest contains one or more syntax errors.';
    Win32ErrorCodes.ERROR_SXS_XML_E_MISSINGQUOTE:
        Win32ErrorCodeDescription := 'Manifest Parse Error : A string literal was expected, but no opening quote character was found.';
    Win32ErrorCodes.ERROR_SXS_XML_E_COMMENTSYNTAX:
        Win32ErrorCodeDescription :=
            'Manifest Parse Error : Incorrect syntax was used in a comment.';
    Win32ErrorCodes.ERROR_SXS_XML_E_BADSTARTNAMECHAR:
        Win32ErrorCodeDescription :=
            'Manifest Parse Error : A name was started with an invalid character.';
    Win32ErrorCodes.ERROR_SXS_XML_E_BADNAMECHAR:
        Win32ErrorCodeDescription :=
            'Manifest Parse Error : A name contained an invalid character.';
    Win32ErrorCodes.ERROR_SXS_XML_E_BADCHARINSTRING:
        Win32ErrorCodeDescription :=
            'Manifest Parse Error : A string literal contained an invalid character.';
    Win32ErrorCodes.ERROR_SXS_XML_E_XMLDECLSYNTAX:
        Win32ErrorCodeDescription :=
            'Manifest Parse Error : Invalid syntax for an XML declaration.';
    Win32ErrorCodes.ERROR_SXS_XML_E_BADCHARDATA:
        Win32ErrorCodeDescription :=
            'Manifest Parse Error : An invalid character was found in text content.';
    Win32ErrorCodes.ERROR_SXS_XML_E_MISSINGWHITESPACE:
        Win32ErrorCodeDescription := 'Manifest Parse Error : Required white space was missing.';
    Win32ErrorCodes.ERROR_SXS_XML_E_EXPECTINGTAGEND:
        Win32ErrorCodeDescription := 'Manifest Parse Error : The character &gt; was expected.';
    Win32ErrorCodes.ERROR_SXS_XML_E_MISSINGSEMICOLON:
        Win32ErrorCodeDescription := 'Manifest Parse Error : A semi colon character was expected.';
    Win32ErrorCodes.ERROR_SXS_XML_E_UNBALANCEDPAREN:
        Win32ErrorCodeDescription := 'Manifest Parse Error : Unbalanced parentheses.';
    Win32ErrorCodes.ERROR_SXS_XML_E_INTERNALERROR:
        Win32ErrorCodeDescription := 'Manifest Parse Error : Internal error.';
    Win32ErrorCodes.ERROR_SXS_XML_E_UNEXPECTED_WHITESPACE:
        Win32ErrorCodeDescription :=
            'Manifest Parse Error : White space is not allowed at this location.';
    Win32ErrorCodes.ERROR_SXS_XML_E_INCOMPLETE_ENCODING:
        Win32ErrorCodeDescription :=
            'Manifest Parse Error : End of file reached in invalid state for current encoding.';
    Win32ErrorCodes.ERROR_SXS_XML_E_MISSING_PAREN:
        Win32ErrorCodeDescription := 'Manifest Parse Error : Missing parenthesis.';
    Win32ErrorCodes.ERROR_SXS_XML_E_EXPECTINGCLOSEQUOTE:
        Win32ErrorCodeDescription :=
            'Manifest Parse Error : A single or double closing quote character (\ or \") is missing.';
    Win32ErrorCodes.ERROR_SXS_XML_E_MULTIPLE_COLONS:
        Win32ErrorCodeDescription :=
            'Manifest Parse Error : Multiple colons are not allowed in a name.';
    Win32ErrorCodes.ERROR_SXS_XML_E_INVALID_DECIMAL:
        Win32ErrorCodeDescription := 'Manifest Parse Error : Invalid character for decimal digit.';
    Win32ErrorCodes.ERROR_SXS_XML_E_INVALID_HEXIDECIMAL:
        Win32ErrorCodeDescription :=
            'Manifest Parse Error : Invalid character for hexadecimal digit.';
    Win32ErrorCodes.ERROR_SXS_XML_E_INVALID_UNICODE:
        Win32ErrorCodeDescription :=
            'Manifest Parse Error : Invalid Unicode character value for this platform.';
    Win32ErrorCodes.ERROR_SXS_XML_E_WHITESPACEORQUESTIONMARK:
        Win32ErrorCodeDescription := 'Manifest Parse Error : Expecting white space or ?.';
    Win32ErrorCodes.ERROR_SXS_XML_E_UNEXPECTEDENDTAG:
        Win32ErrorCodeDescription :=
            'Manifest Parse Error : End tag was not expected at this location.';
    Win32ErrorCodes.ERROR_SXS_XML_E_UNCLOSEDTAG:
        Win32ErrorCodeDescription :=
            'Manifest Parse Error : The following tags were not closed: %1.';
    Win32ErrorCodes.ERROR_SXS_XML_E_DUPLICATEATTRIBUTE:
        Win32ErrorCodeDescription := 'Manifest Parse Error : Duplicate attribute.';
    Win32ErrorCodes.ERROR_SXS_XML_E_MULTIPLEROOTS:
        Win32ErrorCodeDescription :=
            'Manifest Parse Error : Only one top level element is allowed in an XML document.';
    Win32ErrorCodes.ERROR_SXS_XML_E_INVALIDATROOTLEVEL:
        Win32ErrorCodeDescription :=
            'Manifest Parse Error : Invalid at the top level of the document.';
    Win32ErrorCodes.ERROR_SXS_XML_E_BADXMLDECL:
        Win32ErrorCodeDescription := 'Manifest Parse Error : Invalid XML declaration.';
    Win32ErrorCodes.ERROR_SXS_XML_E_MISSINGROOT:
        Win32ErrorCodeDescription :=
            'Manifest Parse Error : XML document must have a top level element.';
    Win32ErrorCodes.ERROR_SXS_XML_E_UNEXPECTEDEOF:
        Win32ErrorCodeDescription := 'Manifest Parse Error : Unexpected end of file.';
    Win32ErrorCodes.ERROR_SXS_XML_E_BADPEREFINSUBSET:
        Win32ErrorCodeDescription := 'Manifest Parse Error : Parameter entities cannot be used inside markup declarations in an internal subset.';
    Win32ErrorCodes.ERROR_SXS_XML_E_UNCLOSEDSTARTTAG:
        Win32ErrorCodeDescription := 'Manifest Parse Error : Element was not closed.';
    Win32ErrorCodes.ERROR_SXS_XML_E_UNCLOSEDENDTAG:
        Win32ErrorCodeDescription :=
            'Manifest Parse Error : End element was missing the character &gt;.';
    Win32ErrorCodes.ERROR_SXS_XML_E_UNCLOSEDSTRING:
        Win32ErrorCodeDescription := 'Manifest Parse Error : A string literal was not closed.';
    Win32ErrorCodes.ERROR_SXS_XML_E_UNCLOSEDCOMMENT:
        Win32ErrorCodeDescription := 'Manifest Parse Error : A comment was not closed.';
    Win32ErrorCodes.ERROR_SXS_XML_E_UNCLOSEDDECL:
        Win32ErrorCodeDescription := 'Manifest Parse Error : A declaration was not closed.';
    Win32ErrorCodes.ERROR_SXS_XML_E_UNCLOSEDCDATA:
        Win32ErrorCodeDescription := 'Manifest Parse Error : A CDATA section was not closed.';
    Win32ErrorCodes.ERROR_SXS_XML_E_RESERVEDNAMESPACE:
        Win32ErrorCodeDescription := 'Manifest Parse Error : The namespace prefix is not allowed to start with the reserved string "xml".';
    Win32ErrorCodes.ERROR_SXS_XML_E_INVALIDENCODING:
        Win32ErrorCodeDescription :=
            'Manifest Parse Error : System does not support the specified encoding.';
    Win32ErrorCodes.ERROR_SXS_XML_E_INVALIDSWITCH:
        Win32ErrorCodeDescription :=
            'Manifest Parse Error : Switch from current encoding to specified encoding not supported.';
    Win32ErrorCodes.ERROR_SXS_XML_E_BADXMLCASE:
        Win32ErrorCodeDescription :=
            'Manifest Parse Error : The name xml is reserved and must be lower case.';
    Win32ErrorCodes.ERROR_SXS_XML_E_INVALID_STANDALONE:
        Win32ErrorCodeDescription :=
            'Manifest Parse Error : The standalone attribute must have the value yes or no.';
    Win32ErrorCodes.ERROR_SXS_XML_E_UNEXPECTED_STANDALONE:
        Win32ErrorCodeDescription :=
            'Manifest Parse Error : The standalone attribute cannot be used in external entities.';
    Win32ErrorCodes.ERROR_SXS_XML_E_INVALID_VERSION:
        Win32ErrorCodeDescription := 'Manifest Parse Error : Invalid version number.';
    Win32ErrorCodes.ERROR_SXS_XML_E_MISSINGEQUALS:
        Win32ErrorCodeDescription :=
            'Manifest Parse Error : Missing equals sign between attribute and attribute value.';
    Win32ErrorCodes.ERROR_IPSEC_QM_POLICY_EXISTS:
        Win32ErrorCodeDescription := 'The specified quick mode policy already exists.';
    Win32ErrorCodes.ERROR_IPSEC_QM_POLICY_NOT_FOUND:
        Win32ErrorCodeDescription := 'The specified quick mode policy was not found.';
    Win32ErrorCodes.ERROR_IPSEC_QM_POLICY_IN_USE:
        Win32ErrorCodeDescription := 'The specified quick mode policy is being used.';
    Win32ErrorCodes.ERROR_IPSEC_MM_POLICY_EXISTS:
        Win32ErrorCodeDescription := 'The specified main mode policy already exists.';
    Win32ErrorCodes.ERROR_IPSEC_MM_POLICY_NOT_FOUND:
        Win32ErrorCodeDescription := 'The specified main mode policy was not found.';
    Win32ErrorCodes.ERROR_IPSEC_MM_POLICY_IN_USE:
        Win32ErrorCodeDescription := 'The specified main mode policy is being used.';
    Win32ErrorCodes.ERROR_IPSEC_MM_FILTER_EXISTS:
        Win32ErrorCodeDescription := 'The specified main mode filter already exists.';
    Win32ErrorCodes.ERROR_IPSEC_MM_FILTER_NOT_FOUND:
        Win32ErrorCodeDescription := 'The specified main mode filter was not found.';
    Win32ErrorCodes.ERROR_IPSEC_TRANSPORT_FILTER_EXISTS:
        Win32ErrorCodeDescription := 'The specified transport mode filter already exists.';
    Win32ErrorCodes.ERROR_IPSEC_TRANSPORT_FILTER_NOT_FOUND:
        Win32ErrorCodeDescription := 'The specified transport mode filter does not exist.';
    Win32ErrorCodes.ERROR_IPSEC_MM_AUTH_EXISTS:
        Win32ErrorCodeDescription := 'The specified main mode authentication list exists.';
    Win32ErrorCodes.ERROR_IPSEC_MM_AUTH_NOT_FOUND:
        Win32ErrorCodeDescription := 'The specified main mode authentication list was not found.';
    Win32ErrorCodes.ERROR_IPSEC_MM_AUTH_IN_USE:
        Win32ErrorCodeDescription := 'The specified quick mode policy is being used.';
    Win32ErrorCodes.ERROR_IPSEC_DEFAULT_MM_POLICY_NOT_FOUND:
        Win32ErrorCodeDescription := 'The specified main mode policy was not found.';
    Win32ErrorCodes.ERROR_IPSEC_DEFAULT_MM_AUTH_NOT_FOUND:
        Win32ErrorCodeDescription := 'The specified quick mode policy was not found.';
    Win32ErrorCodes.ERROR_IPSEC_DEFAULT_QM_POLICY_NOT_FOUND:
        Win32ErrorCodeDescription := 'The manifest file contains one or more syntax errors.';
    Win32ErrorCodes.ERROR_IPSEC_TUNNEL_FILTER_EXISTS:
        Win32ErrorCodeDescription :=
            'The application attempted to activate a disabled activation context.';
    Win32ErrorCodes.ERROR_IPSEC_TUNNEL_FILTER_NOT_FOUND:
        Win32ErrorCodeDescription :=
            'The requested lookup key was not found in any active activation context.';
    Win32ErrorCodes.ERROR_IPSEC_MM_FILTER_PENDING_DELETION:
        Win32ErrorCodeDescription := 'The Main Mode filter is pending deletion.';
    Win32ErrorCodes.ERROR_IPSEC_TRANSPORT_FILTER_PENDING_DELETION:
        Win32ErrorCodeDescription := 'The transport filter is pending deletion.';
    Win32ErrorCodes.ERROR_IPSEC_TUNNEL_FILTER_PENDING_DELETION:
        Win32ErrorCodeDescription := 'The tunnel filter is pending deletion.';
    Win32ErrorCodes.ERROR_IPSEC_MM_POLICY_PENDING_DELETION:
        Win32ErrorCodeDescription := 'The Main Mode policy is pending deletion.';
    Win32ErrorCodes.ERROR_IPSEC_MM_AUTH_PENDING_DELETION:
        Win32ErrorCodeDescription := 'The Main Mode authentication bundle is pending deletion.';
    Win32ErrorCodes.ERROR_IPSEC_QM_POLICY_PENDING_DELETION:
        Win32ErrorCodeDescription := 'The Quick Mode policy is pending deletion.';
    Win32ErrorCodes.ERROR_IPSEC_IKE_AUTH_FAIL:
        Win32ErrorCodeDescription := 'IKE authentication credentials are unacceptable.';
    Win32ErrorCodes.ERROR_IPSEC_IKE_ATTRIB_FAIL:
        Win32ErrorCodeDescription := 'IKE security attributes are unacceptable.';
    Win32ErrorCodes.ERROR_IPSEC_IKE_NEGOTIATION_PENDING:
        Win32ErrorCodeDescription := 'IKE Negotiation in progress.';
    Win32ErrorCodes.ERROR_IPSEC_IKE_GENERAL_PROCESSING_ERROR:
        Win32ErrorCodeDescription := 'General processing error.';
    Win32ErrorCodes.ERROR_IPSEC_IKE_TIMED_OUT:
        Win32ErrorCodeDescription := 'Negotiation timed out.';
    Win32ErrorCodes.ERROR_IPSEC_IKE_NO_CERT:
        Win32ErrorCodeDescription := 'IKE failed to find valid machine certificate.';
    Win32ErrorCodes.ERROR_IPSEC_IKE_SA_DELETED:
        Win32ErrorCodeDescription := 'IKE SA deleted by peer before establishment completed.';
    Win32ErrorCodes.ERROR_IPSEC_IKE_SA_REAPED:
        Win32ErrorCodeDescription := 'IKE SA deleted before establishment completed.';
    Win32ErrorCodes.ERROR_IPSEC_IKE_MM_ACQUIRE_DROP:
        Win32ErrorCodeDescription := 'Negotiation request sat in Queue too long.';
    Win32ErrorCodes.ERROR_IPSEC_IKE_QM_ACQUIRE_DROP:
        Win32ErrorCodeDescription := 'Negotiation request sat in Queue too long.';
    Win32ErrorCodes.ERROR_IPSEC_IKE_QUEUE_DROP_MM:
        Win32ErrorCodeDescription := 'Negotiation request sat in Queue too long.';
    Win32ErrorCodes.ERROR_IPSEC_IKE_QUEUE_DROP_NO_MM:
        Win32ErrorCodeDescription := 'Negotiation request sat in Queue too long.';
    Win32ErrorCodes.ERROR_IPSEC_IKE_DROP_NO_RESPONSE:
        Win32ErrorCodeDescription := 'No response from peer.';
    Win32ErrorCodes.ERROR_IPSEC_IKE_MM_DELAY_DROP:
        Win32ErrorCodeDescription := 'Negotiation took too long.';
    Win32ErrorCodes.ERROR_IPSEC_IKE_QM_DELAY_DROP:
        Win32ErrorCodeDescription := 'Negotiation took too long.';
    Win32ErrorCodes.ERROR_IPSEC_IKE_ERROR:
        Win32ErrorCodeDescription := 'Unknown error occurred.';
    Win32ErrorCodes.ERROR_IPSEC_IKE_CRL_FAILED:
        Win32ErrorCodeDescription := 'Certificate Revocation Check failed.';
    Win32ErrorCodes.ERROR_IPSEC_IKE_INVALID_KEY_USAGE:
        Win32ErrorCodeDescription := 'Invalid certificate key usage.';
    Win32ErrorCodes.ERROR_IPSEC_IKE_INVALID_CERT_TYPE:
        Win32ErrorCodeDescription := 'Invalid certificate type.';
    Win32ErrorCodes.ERROR_IPSEC_IKE_NO_PRIVATE_KEY:
        Win32ErrorCodeDescription := 'No private key associated with machine certificate.';
    Win32ErrorCodes.ERROR_IPSEC_IKE_DH_FAIL:
        Win32ErrorCodeDescription := 'Failure in Diffie-Helman computation.';
    Win32ErrorCodes.ERROR_IPSEC_IKE_INVALID_HEADER:
        Win32ErrorCodeDescription := 'Invalid header.';
    Win32ErrorCodes.ERROR_IPSEC_IKE_NO_POLICY:
        Win32ErrorCodeDescription := 'No policy configured.';
    Win32ErrorCodes.ERROR_IPSEC_IKE_INVALID_SIGNATURE:
        Win32ErrorCodeDescription := 'Failed to verify signature.';
    Win32ErrorCodes.ERROR_IPSEC_IKE_KERBEROS_ERROR:
        Win32ErrorCodeDescription := 'Failed to authenticate using Kerberos.';
    Win32ErrorCodes.ERROR_IPSEC_IKE_NO_PUBLIC_KEY:
        Win32ErrorCodeDescription := 'Peers certificate did not have a public key.';
    Win32ErrorCodes.ERROR_IPSEC_IKE_PROCESS_ERR:
        Win32ErrorCodeDescription := 'Error processing error payload.';
    Win32ErrorCodes.ERROR_IPSEC_IKE_PROCESS_ERR_SA:
        Win32ErrorCodeDescription := 'Error processing SA payload.';
    Win32ErrorCodes.ERROR_IPSEC_IKE_PROCESS_ERR_PROP:
        Win32ErrorCodeDescription := 'Error processing Proposal payload.';
    Win32ErrorCodes.ERROR_IPSEC_IKE_PROCESS_ERR_TRANS:
        Win32ErrorCodeDescription := 'Error processing Transform payload.';
    Win32ErrorCodes.ERROR_IPSEC_IKE_PROCESS_ERR_KE:
        Win32ErrorCodeDescription := 'Error processing KE payload.';
    Win32ErrorCodes.ERROR_IPSEC_IKE_PROCESS_ERR_ID:
        Win32ErrorCodeDescription := 'Error processing ID payload.';
    Win32ErrorCodes.ERROR_IPSEC_IKE_PROCESS_ERR_CERT:
        Win32ErrorCodeDescription := 'Error processing Cert payload.';
    Win32ErrorCodes.ERROR_IPSEC_IKE_PROCESS_ERR_CERT_REQ:
        Win32ErrorCodeDescription := 'Error processing Certificate Request payload.';
    Win32ErrorCodes.ERROR_IPSEC_IKE_PROCESS_ERR_HASH:
        Win32ErrorCodeDescription := 'Error processing Hash payload.';
    Win32ErrorCodes.ERROR_IPSEC_IKE_PROCESS_ERR_SIG:
        Win32ErrorCodeDescription := 'Error processing Signature payload.';
    Win32ErrorCodes.ERROR_IPSEC_IKE_PROCESS_ERR_NONCE:
        Win32ErrorCodeDescription := 'Error processing Nonce payload.';
    Win32ErrorCodes.ERROR_IPSEC_IKE_PROCESS_ERR_NOTIFY:
        Win32ErrorCodeDescription := 'Error processing Notify payload.';
    Win32ErrorCodes.ERROR_IPSEC_IKE_PROCESS_ERR_DELETE:
        Win32ErrorCodeDescription := 'Error processing Delete Payload.';
    Win32ErrorCodes.ERROR_IPSEC_IKE_PROCESS_ERR_VENDOR:
        Win32ErrorCodeDescription := 'Error processing VendorId payload.';
    Win32ErrorCodes.ERROR_IPSEC_IKE_INVALID_PAYLOAD:
        Win32ErrorCodeDescription := 'Invalid payload received.';
    Win32ErrorCodes.ERROR_IPSEC_IKE_LOAD_SOFT_SA:
        Win32ErrorCodeDescription := 'Soft SA loaded.';
    Win32ErrorCodes.ERROR_IPSEC_IKE_SOFT_SA_TORN_DOWN:
        Win32ErrorCodeDescription := 'Soft SA torn down.';
    Win32ErrorCodes.ERROR_IPSEC_IKE_INVALID_COOKIE:
        Win32ErrorCodeDescription := 'Invalid cookie received..';
    Win32ErrorCodes.ERROR_IPSEC_IKE_NO_PEER_CERT:
        Win32ErrorCodeDescription := 'Peer failed to send valid machine certificate.';
    Win32ErrorCodes.ERROR_IPSEC_IKE_PEER_CRL_FAILED:
        Win32ErrorCodeDescription := 'Certification Revocation check of peers certificate failed.';
    Win32ErrorCodes.ERROR_IPSEC_IKE_POLICY_CHANGE:
        Win32ErrorCodeDescription := 'New policy invalidated SAs formed with old policy.';
    Win32ErrorCodes.ERROR_IPSEC_IKE_NO_MM_POLICY:
        Win32ErrorCodeDescription := 'There is no available Main Mode IKE policy.';
    Win32ErrorCodes.ERROR_IPSEC_IKE_NOTCBPRIV:
        Win32ErrorCodeDescription := 'Failed to enabled TCB privilege.';
    Win32ErrorCodes.ERROR_IPSEC_IKE_SECLOADFAIL:
        Win32ErrorCodeDescription := 'Failed to load SECURITY.DLL.';
    Win32ErrorCodes.ERROR_IPSEC_IKE_FAILSSPINIT:
        Win32ErrorCodeDescription :=
            'Failed to obtain security function table dispatch address from SSPI.';
    Win32ErrorCodes.ERROR_IPSEC_IKE_FAILQUERYSSP:
        Win32ErrorCodeDescription := 'Failed to query Kerberos package to obtain max token size.';
    Win32ErrorCodes.ERROR_IPSEC_IKE_SRVACQFAIL:
        Win32ErrorCodeDescription := 'Failed to obtain Kerberos server credentials for ISAKMP/ERROR_IPSEC_IKE service. Kerberos authentication will not function. The most likely reason for this is lack of domain membership. This is normal if your computer is a member of a workgroup.';
    Win32ErrorCodes.ERROR_IPSEC_IKE_SRVQUERYCRED:
        Win32ErrorCodeDescription := 'Failed to determine SSPI principal name for ISAKMP/ERROR_IPSEC_IKE service (QueryCredentialsAttributes).';
    Win32ErrorCodes.ERROR_IPSEC_IKE_GETSPIFAIL:
        Win32ErrorCodeDescription := 'Failed to obtain new SPI for the inbound SA from Ipsec driver. The most common cause for this is that the driver does not have the correct filter. Check your policy to verify the filters.';
    Win32ErrorCodes.ERROR_IPSEC_IKE_INVALID_FILTER:
        Win32ErrorCodeDescription := 'Given filter is invalid.';
    Win32ErrorCodes.ERROR_IPSEC_IKE_OUT_OF_MEMORY:
        Win32ErrorCodeDescription := 'Memory allocation failed.';
    Win32ErrorCodes.ERROR_IPSEC_IKE_ADD_UPDATE_KEY_FAILED:
        Win32ErrorCodeDescription := 'Failed to add Security Association to IPSec Driver. The most common cause for this is if the IKE negotiation took too long to complete. If the problem persists, reduce the load on the faulting machine.';
    Win32ErrorCodes.ERROR_IPSEC_IKE_INVALID_POLICY:
        Win32ErrorCodeDescription := 'Invalid policy.';
    Win32ErrorCodes.ERROR_IPSEC_IKE_UNKNOWN_DOI:
        Win32ErrorCodeDescription := 'Invalid DOI.';
    Win32ErrorCodes.ERROR_IPSEC_IKE_INVALID_SITUATION:
        Win32ErrorCodeDescription := 'Invalid situation.';
    Win32ErrorCodes.ERROR_IPSEC_IKE_DH_FAILURE:
        Win32ErrorCodeDescription := 'Diffie-Hellman failure.';
    Win32ErrorCodes.ERROR_IPSEC_IKE_INVALID_GROUP:
        Win32ErrorCodeDescription := 'Invalid Diffie-Hellman group.';
    Win32ErrorCodes.ERROR_IPSEC_IKE_ENCRYPT:
        Win32ErrorCodeDescription := 'Error encrypting payload.';
    Win32ErrorCodes.ERROR_IPSEC_IKE_DECRYPT:
        Win32ErrorCodeDescription := 'Error decrypting payload.';
    Win32ErrorCodes.ERROR_IPSEC_IKE_POLICY_MATCH:
        Win32ErrorCodeDescription := 'Policy match error.';
    Win32ErrorCodes.ERROR_IPSEC_IKE_UNSUPPORTED_ID:
        Win32ErrorCodeDescription := 'Unsupported ID.';
    Win32ErrorCodes.ERROR_IPSEC_IKE_INVALID_HASH:
        Win32ErrorCodeDescription := 'Hash verification failed.';
    Win32ErrorCodes.ERROR_IPSEC_IKE_INVALID_HASH_ALG:
        Win32ErrorCodeDescription := 'Invalid hash algorithm.';
    Win32ErrorCodes.ERROR_IPSEC_IKE_INVALID_HASH_SIZE:
        Win32ErrorCodeDescription := 'Invalid hash size.';
    Win32ErrorCodes.ERROR_IPSEC_IKE_INVALID_ENCRYPT_ALG:
        Win32ErrorCodeDescription := 'Invalid encryption algorithm.';
    Win32ErrorCodes.ERROR_IPSEC_IKE_INVALID_AUTH_ALG:
        Win32ErrorCodeDescription := 'Invalid authentication algorithm.';
    Win32ErrorCodes.ERROR_IPSEC_IKE_INVALID_SIG:
        Win32ErrorCodeDescription := 'Invalid certificate signature.';
    Win32ErrorCodes.ERROR_IPSEC_IKE_LOAD_FAILED:
        Win32ErrorCodeDescription := 'Load failed.';
    Win32ErrorCodes.ERROR_IPSEC_IKE_RPC_DELETE:
        Win32ErrorCodeDescription := 'Deleted via RPC call.';
    Win32ErrorCodes.ERROR_IPSEC_IKE_BENIGN_REINIT:
        Win32ErrorCodeDescription :=
            'Temporary state created to perform reinitialization. This is not a real failure.';
    Win32ErrorCodes.ERROR_IPSEC_IKE_INVALID_RESPONDER_LIFETIME_NOTIFY:
        Win32ErrorCodeDescription := 'The lifetime value received in the Responder Lifetime Notify is below the Windows 2000 configured minimum value. Please fix the policy on the peer machine.';
    Win32ErrorCodes.ERROR_IPSEC_IKE_QM_LIMIT_REAP:
        Win32ErrorCodeDescription := 'SA reaped because QM limit was reached.';
    Win32ErrorCodes.ERROR_IPSEC_IKE_INVALID_CERT_KEYLEN:
        Win32ErrorCodeDescription :=
            'Key length in certificate is too small for configured security requirements.';
    Win32ErrorCodes.ERROR_IPSEC_IKE_MM_LIMIT:
        Win32ErrorCodeDescription := 'Max number of established MM SAs to peer exceeded.';
    Win32ErrorCodes.ERROR_IPSEC_IKE_NEGOTIATION_DISABLED:
        Win32ErrorCodeDescription := 'IKE received a policy that disables negotiation.';
    Win32ErrorCodes.ERROR_IPSEC_IKE_QM_LIMIT:
        Win32ErrorCodeDescription :=
            'Reached maximum quick mode limit for the main mode. New main mode will be started.';
ELSE
    Win32ErrorCodeDescription := 'Unknown Win32 error code.';
END_CASE

END_FUNCTION

// Win32_Tests/ToWin32ErrorCode_Tests
{attribute 'hide'}
FUNCTION_BLOCK ToWin32ErrorCode_Tests EXTENDS TcUnit.FB_TestSuite

ConversionOfValidErrorCode();
ConversionOfInvalidErrorCode();

METHOD ConversionOfInvalidErrorCode
TcUnit.TEST('ConversionOfInvalidErrorCode');

AssertEquals_UDINT(
    Expected:=Win32ErrorCodes.ERR_UNKNOWN,
    Actual:=ToWin32ErrorCode(1234567),
    Message:='Error conversion not correct.'
);

TcUnit.TEST_FINISHED();
END_METHOD

METHOD ConversionOfValidErrorCode
TcUnit.TEST('ConversionOfValidErrorCode');

AssertEquals_UDINT(
    Expected:=Win32ErrorCodes.ERROR_FILE_EXISTS,
    Actual:=ToWin32ErrorCode(80),
    Message:='Error conversion not correct.'
);

TcUnit.TEST_FINISHED();
END_METHOD

END_FUNCTION_BLOCK

// Win32_Tests/Win32ErrorCodeDesciption_Tests
{attribute 'hide'}
FUNCTION_BLOCK Win32ErrorCodeDesciption_Tests EXTENDS TcUnit.FB_TestSuite

DescriptionOfKnownErrorCode();
DescriptionOfUnknownErrorCode();

METHOD DescriptionOfKnownErrorCode
TcUnit.TEST('DescriptionOfKnownErrorCode');

AssertEquals_STRING(
    Expected:='The system cannot find the file specified.',
    Actual:=Win32ErrorCodeDescription(Win32ErrorCodes.ERROR_FILE_NOT_FOUND),
    Message:='Error description not correct.'
);

TcUnit.TEST_FINISHED();
END_METHOD

METHOD DescriptionOfUnknownErrorCode
TcUnit.TEST('DescriptionOfUnknownErrorCode');

AssertEquals_STRING(
    Expected:='Unknown Win32 error code.',
    Actual:=Win32ErrorCodeDescription(Win32ErrorCodes.ERR_UNKNOWN),
    Message:='Error description not correct.'
);

TcUnit.TEST_FINISHED();
END_METHOD

END_FUNCTION_BLOCK

// UnitTests
{attribute 'hide'}
PROGRAM UnitTests
VAR
    {attribute 'analysis' := '-33'}
    toWin32ErrorCode_Tests : ToWin32ErrorCode_Tests;
    {attribute 'analysis' := '-33'}
    win32ErrorCodeDescription_Tests : Win32ErrorCodeDesciption_Tests;
END_VAR

TcUnit.RUN();

END_PROGRAM
